FUNCTION_BLOCK PUBLIC ABSTRACT Cyclic_Task_Base
VAR
	_busy : BOOL;
	_error : BOOL;
	_done : BOOL;
END_VAR

METHOD Abort : BOOL
VAR_INPUT
END_VAR
END_METHOD

PROPERTY Busy : bool
GET
Busy := _busy;
END_GET
END_PROPERTY

METHOD Cycle : BOOL
VAR_INPUT
END_VAR
END_METHOD

PROPERTY Done : bool
GET
Done := _done;
END_GET
END_PROPERTY

PROPERTY Error : bool
GET
Error := _error;
END_GET
END_PROPERTY

END_FUNCTION_BLOCK

(* stored: Version 1.1.0.1, ProductVersion 3.1.4024.11
   POU Cyclic_Task_Base: Id {39e04cde-e357-4b4d-b156-8fa2608de0da}, SpecialFunc None
   Method Abort: Id {e3c8f471-9e76-486d-ad1c-9581b8fb752c}
   Property Busy: Id {530dd4f8-a224-4247-831b-b8b5a7454280}
   Get Get: Id {ebf38750-9bf5-469e-a2c9-45e1cfd30637}
   Method Cycle: Id {2948c0cf-06e0-464b-88b4-99d13f08064e}
   Property Done: Id {8c5f6e53-0be8-47f9-a497-fde2f525545a}
   Get Get: Id {7796751c-3390-4541-bb0a-d232fd124f45}
   Property Error: Id {617deeb8-6775-483e-87db-21bff7368ee6}
   Get Get: Id {e0e82b73-eb33-45ef-b31b-843731fff403} *)
